FUNCTION_BLOCK EVENT_ANALYZER
  {SET_ATTRIBUTE(OpcUa, SERVICE)}
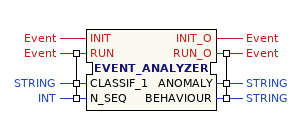
  EVENT_INPUT
    INIT;
    RUN WITH CLASSIF_1, N_SEQ; {SET_ATTRIBUTE(OpcUa, Method)}
  END_EVENT
  EVENT_OUTPUT
    INIT_O;
    RUN_O WITH ANOMALY, BEHAVIOUR;
  END_EVENT
  VAR_INPUT
    CLASSIF_1 : STRING; {SET_ATTRIBUTE(OpcUa, Variable.RUN)}
    N_SEQ : INT; {SET_ATTRIBUTE(OpcUa, Variable.RUN)}
  END_VAR
  VAR_OUTPUT
    ANOMALY : STRING; {SET_ATTRIBUTE(OpcUa, Variable.RUN)}
    BEHAVIOUR : STRING; {SET_ATTRIBUTE(OpcUa, Variable.RUN)}
  END_VAR
END_FUNCTION_BLOCK
